(* 
:Description: This function block allows to log the data to the buffer
*)
FUNCTION_BLOCK FB_Buffer
VAR
	sName 			: STRING;
	MAX_BUFFER_SIZE : UDINT;
	arrBuffer 		: ARRAY[0..MAX_BUFFER_SIZE] OF BYTE; (* Buffer memory used by FB_MemRingBuffer function block *)
	
	(* Internal status *)
	bActive 					: BOOL;						(*  *)
	bBusy						: BOOL;						(*  *)
	bError						: BOOL;						(*  *)
	iErrorID					: UDINT;					(*  *)
	
	(* Function blocks - buffer handling *)
	fbBuffer					: FB_MemRingBuffer;
	
	(* State machines *)
	eBufferState				: E_BufferState;
	eBufferInitState			: E_BufferInitState;
END_VAR

PROPERTY Active : REFERENCE TO BOOL
GET
Active REF= bActive;
END_GET
END_PROPERTY

PROPERTY Busy : REFERENCE TO BOOL
GET
Busy REF= bBusy;
END_GET
END_PROPERTY

PROPERTY Error : REFERENCE TO BOOL
GET
Error REF= bError;
END_GET
END_PROPERTY

PROPERTY ErrorID : REFERENCE TO UDINT
GET
ErrorID REF= iErrorID;
END_GET
END_PROPERTY

METHOD MR_FirstCycle : BOOL
VAR_INPUT
	sName 			: STRING;
	MAX_BUFFER_SIZE : UDINT;
	
END_VAR
THIS^.sName := sName;
THIS^.MAX_BUFFER_SIZE := MAX_BUFFER_SIZE;
END_METHOD

METHOD MR_Init : BOOL
VAR_INPUT
END_VAR
IF eBufferState = BUFFER_UNINITIALIZED THEN
	bBusy := TRUE;
	MR_Init := FALSE;
	eBufferState := BUFFER_INITIALIZING;
	
ELSIF eBufferState := BUFFER_READY THEN
	bBusy := FALSE;
	MR_Init := TRUE;
	
END_IF
END_METHOD

METHOD PROTECTED MS_Initializing
CASE eBufferInitState OF
	
END_CASE
END_METHOD

METHOD PROTECTED MS_Uninitialized
;
END_METHOD

METHOD PROTECTED StateMachine : BOOL
VAR_INPUT
END_VAR
CASE eBufferState OF
	BUFFER_UNINITIALIZED:
		MS_Uninitialized();
	
	BUFFER_INITIALIZING:
		
END_CASE
END_METHOD

END_FUNCTION_BLOCK

(* stored: Version 1.1.0.1, ProductVersion 3.1.4024.9
   POU FB_Buffer: Id {bfe92a21-68c0-4c91-91d9-ceb661de1969}, SpecialFunc None
   Folder FirstCycle: Id {c0cb9efa-c63a-44dc-aac0-560412c22bee}
   Folder Properties: Id {50b54840-c606-4efe-9e99-fcadc7c53e33}
   Folder Requests: Id {345e277a-0100-4003-96d4-1fd6f7358b4d}
   Folder StateMachine: Id {3c1c347f-176d-491a-9618-1a847225048c}
   Property Active: Id {68ee4ceb-b0b5-4544-a166-6f570644d20b}
   Get Get: Id {0b8e58c5-a4de-4dc0-8ec0-fa5cc21507c2}
   Property Busy: Id {687a8547-e55c-48b7-9f56-e0d843c2f4ce}
   Get Get: Id {3d982172-8c1a-49f8-b57d-863b054c4964}
   Property Error: Id {da746dad-1602-4a9e-b81f-03189b4eb9a9}
   Get Get: Id {b05c7773-deaf-4881-a79e-5256802f6113}
   Property ErrorID: Id {94845ebf-176e-4701-946b-f3173952c32c}
   Get Get: Id {743f855e-29be-48f6-8f34-ac08caa835e5}
   Method MR_FirstCycle: Id {4a615ef0-caa0-4488-8eb5-5de764d7cc9d}
   Method MR_Init: Id {96faae37-bed6-4137-b54a-ac9f4f6e0385}
   Method MS_Initializing: Id {2fa15528-8c84-4c0b-a540-312cad747155}
   Method MS_Uninitialized: Id {6ef825a8-4ef9-465c-a57b-2ecb353a3e15}
   Method StateMachine: Id {0b98d0b0-309d-4e58-bec9-df982c0676a6} *)
